// TIA Portal project "Project1" (V16)

(* hardware
DEVICE "S7-1200 station_1"  S7-1200 Station
   slot 0: "Rack_0"  S7-1200 Rack  Rack  V1.0
   slot 1: "plc_2"  CPU 1214C DC/DC/DC  6ES7 214-1AG40-0XB0  V4.4
   slot 2: "AI 4x13BIT_1"  6ES7 231-4HD32-0XB0  V2.1
   slot 3: "CB 1241 (RS485)"  CB 1241 (RS485)  6ES7 241-1CH30-1XB0  V1.0
*)

// ===== PLC "plc_2"  CPU 1214C DC/DC/DC =====

VAR_GLOBAL   // PLC tag table "Default tag table"
   "System_Byte" AT %MB1 : Byte;
   "FirstScan" AT %M1.0 : Bool;
   "DiagStatusUpdate" AT %M1.1 : Bool;
   "AlwaysTRUE" AT %M1.2 : Bool;
   "AlwaysFALSE" AT %M1.3 : Bool;
   "Clock_Byte" AT %MB0 : Byte;
   "Clock_10Hz" AT %M0.0 : Bool;
   "Clock_5Hz" AT %M0.1 : Bool;
   "Clock_2.5Hz" AT %M0.2 : Bool;
   "Clock_2Hz" AT %M0.3 : Bool;
   "Clock_1.25Hz" AT %M0.4 : Bool;
   "Clock_1Hz" AT %M0.5 : Bool;
   "Clock_0.625Hz" AT %M0.6 : Bool;
   "Clock_0.5Hz" AT %M0.7 : Bool;
   "RUNNING" AT %M8.1 : Bool;
   "ALARM" AT %M8.2 : Bool;
   "WARNING" AT %M8.3 : Bool;
   "SPEED_VFD" AT %MD10 : Real;
   "CURRENT" AT %MD14 : Real;
   "POWER" AT %MD18 : Real;
   "CARD_TEMPERATURE" AT %IW22 : Int;
   "AI1" AT %MD26 : Real;
   "AI2" AT %MD30 : Real;
   "ALARM_CODE" AT %MW2 : Int;
END_VAR

DATA_BLOCK "Data_block_1"   // DB3
{ S7_Optimized_Access := 'TRUE' }
VERSION : 0.1
   VAR RETAIN
      reference_retain : Real;
   END_VAR
   VAR
      reference_no_retain : Real;
   END_VAR
   VAR RETAIN
      reference_select : Bool;   // wybór pomiędzy zmienną zapamiętywaną po utracie zasilania a zwykłą zmienną
      start_stop_retain : Bool;
   END_VAR
   VAR
      start_stop_no_retain : Bool;
   END_VAR
   VAR RETAIN
      start_stop_select : Bool;   // wybór pomiędzy zmienną zapamiętywaną po utracie zasilania a zwykłą zmienną
   END_VAR
   VAR
      REFERENCE_TO_VFD : Real;
      START_STOP_TO_VFD : Bool;
   END_VAR
BEGIN
END_DATA_BLOCK

// folder: DANFOSS_FC_202

DATA_BLOCK "DB_1_DANFOSS_FC_202"   // DB1
{ S7_Optimized_Access := 'FALSE' }
VERSION : 0.1
   VAR
      reference : Int;
      speed_vfd : Int;
      command : Word;
      current : DInt;
      power : DInt;
      card_temperature : Int;
      AI1 : DInt;
      AI2 : DInt;
      alarm : Bool;
      warning : Bool;
      status : Array[0..15] of Bool;
      alarm_code : UInt;
      alarm_code_array_index : Int := 0;
   END_VAR
BEGIN
   // status[0] : Coil 41, TRUE - At reference, FALSE - Not at reference
   // status[1] : Coil 42, TRUE - Auto mode, FALSE - Hand mode
   // status[2] : Coil 43, TRUE - In frequency range, FALSE - Out of frequency range
   // status[3] : Coil 44, TRUE - Running, FALSE - Stopped
   // status[4] : Coil 45, Not used
   // status[5] : Coil 46, TRUE - Voltage warning, FALSE - No voltage warning
   // status[6] : Coil 47, TRUE - Current limit, FALSE - Not in current limit
   // status[7] : Coil 48, TRUE - Thermal warning, FALSE - No thermal warning
   // status[8] : Coil 33, TRUE - Control ready, FALSE - Control not ready
   // status[9] : Coil 34, TRUE - Frequency converter ready, FALSE - Frequency converter not ready
   // status[10] : Coil 35, TRUE - Safety closed, FALSE - Coasting stop
   // status[11] : Coil 36, TRUE - Alarm, FALSE - No alarm
   // status[12] : Coil 37, Not used
   // status[13] : Coil 38, Not used
   // status[14] : Coil 39, Not used
   // status[15] : Coil 40, TRUE - Warning, FALSE - No warning
END_DATA_BLOCK

// folder: System blocks/Program resources

DATA_BLOCK "IEC_Counter_0_DB"   // DB2
{ S7_Optimized_Access := 'TRUE' }
AUTHOR : Simatic
FAMILY : IEC
NAME : CNTR
VERSION : 1.0
// stored: InstanceOfName IEC_COUNTER
"IEC_COUNTER"
BEGIN
END_DATA_BLOCK

// folder: (top level)

ORGANIZATION_BLOCK "Main"   // OB1, LAD, ProgramCycle
TITLE = "Main Program Sweep (Cycle)"
{ S7_Optimized_Access := 'TRUE' }
VERSION : 0.1
   VAR_INPUT
      Initial_Call : Bool;   // Initial call of this OB
      Remanence : Bool;   // =True, if remanent data are available
   END_VAR
   VAR CONSTANT
      MODBUS_ADRESS : Int := 1;
   END_VAR
BEGIN

REGION Network 1
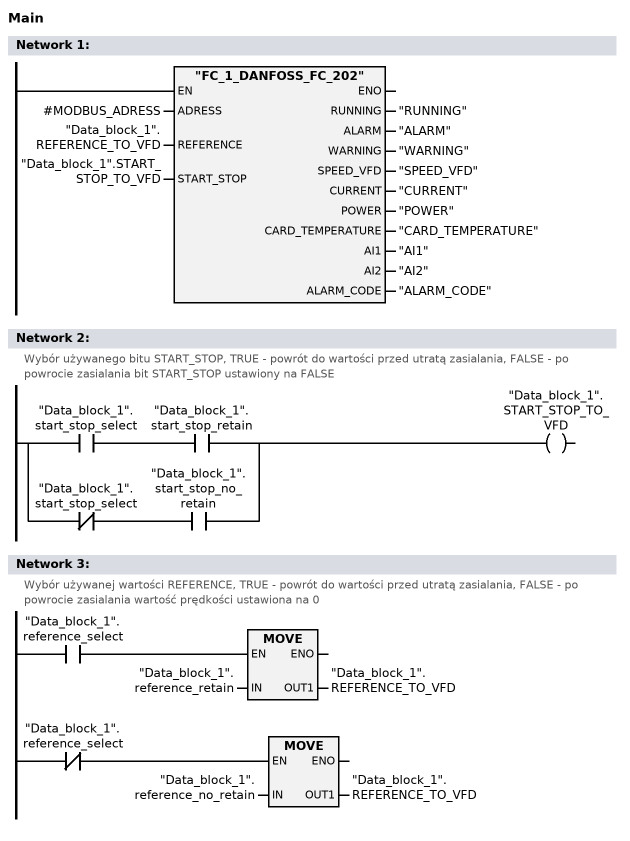
   RUNG wire#powerrail
      "FC_1_DANFOSS_FC_202"(ADRESS := #MODBUS_ADRESS, REFERENCE := "Data_block_1".REFERENCE_TO_VFD, START_STOP := "Data_block_1".START_STOP_TO_VFD, RUNNING => "RUNNING", ALARM => "ALARM", WARNING => "WARNING", SPEED_VFD => "SPEED_VFD", CURRENT => "CURRENT", POWER => "POWER", CARD_TEMPERATURE => "CARD_TEMPERATURE", AI1 => "AI1", AI2 => "AI2", ALARM_CODE => "ALARM_CODE")
   END_RUNG
   // the same network as SCL:
   "FC_1_DANFOSS_FC_202"(ADRESS := #MODBUS_ADRESS,
                         REFERENCE := "Data_block_1".REFERENCE_TO_VFD,
                         START_STOP := "Data_block_1".START_STOP_TO_VFD,
                         RUNNING => "RUNNING",
                         ALARM => "ALARM",
                         WARNING => "WARNING",
                         SPEED_VFD => "SPEED_VFD",
                         CURRENT => "CURRENT",
                         POWER => "POWER",
                         CARD_TEMPERATURE => "CARD_TEMPERATURE",
                         AI1 => "AI1",
                         AI2 => "AI2",
                         ALARM_CODE => "ALARM_CODE");
END_REGION

REGION Network 2
   // Wybór używanego bitu START_STOP, TRUE - powrót do wartości przed utratą zasialania, FALSE - po powrocie zasialania bit START_STOP ustawiony na FALSE
   RUNG wire#powerrail
      Contact( "Data_block_1".start_stop_select )
      Contact( "Data_block_1".start_stop_retain )
      wire#w1
      Coil( "Data_block_1".START_STOP_TO_VFD )
   END_RUNG
   RUNG wire#powerrail
      I_Contact( "Data_block_1".start_stop_select )
      Contact( "Data_block_1".start_stop_no_retain )
   END_RUNG wire#w1
   // the same network as SCL:
   "Data_block_1".START_STOP_TO_VFD := ("Data_block_1".start_stop_select AND "Data_block_1".start_stop_retain) OR (NOT "Data_block_1".start_stop_select AND "Data_block_1".start_stop_no_retain);
END_REGION

REGION Network 3
   // Wybór używanej wartości REFERENCE, TRUE - powrót do wartości przed utratą zasialania, FALSE - po powrocie zasialania wartość prędkości ustawiona na 0
   RUNG wire#powerrail
      Contact( "Data_block_1".reference_select )
      Move(in := "Data_block_1".reference_retain, out1 => "Data_block_1".REFERENCE_TO_VFD)
   END_RUNG
   RUNG wire#powerrail
      I_Contact( "Data_block_1".reference_select )
      Move(in := "Data_block_1".reference_no_retain, out1 => "Data_block_1".REFERENCE_TO_VFD)
   END_RUNG
   // the same network as SCL:
   IF "Data_block_1".reference_select THEN
       "Data_block_1".REFERENCE_TO_VFD := "Data_block_1".reference_retain;
   END_IF;
   IF NOT "Data_block_1".reference_select THEN
       "Data_block_1".REFERENCE_TO_VFD := "Data_block_1".reference_no_retain;
   END_IF;
END_REGION
END_ORGANIZATION_BLOCK

// folder: DANFOSS_FC_202

FUNCTION "FC_1_DANFOSS_FC_202" : Void   // FC1, LAD
{ S7_Optimized_Access := 'TRUE' }
VERSION : 0.1
   VAR_INPUT
      ADRESS : Word;   // address for the frequency converter (standard) port
      REFERENCE : Real;   // frequency 0 - 50 [Hz]
      START_STOP : Bool;   // TRUE - start, FALSE - ramp stop
   END_VAR
   VAR_OUTPUT
      RUNNING : Bool;   // TRUE - Running, FALSE - Stopped
      ALARM : Bool;   // TRUE - Alarm, FALSE - No alarm
      WARNING : Bool;   // TRUE - Warning, FALSE - No warning
      SPEED_VFD : Real;   // frequency [Hz]
      CURRENT : Real;   // current [A]
      POWER : Real;   // power [kW]
      CARD_TEMPERATURE : Int;   // control card temperarue [°C]
      AI1 : Real;   // analog input 1
      AI2 : Real;   // analog input 2
      ALARM_CODE : Int;   // the most recent logged alarm (index 0) from alarm log
   END_VAR
   VAR_TEMP
      tCommand : Word;
      tReference : Real;
      tSpeed : Real;
   END_VAR
BEGIN

REGION Network 1
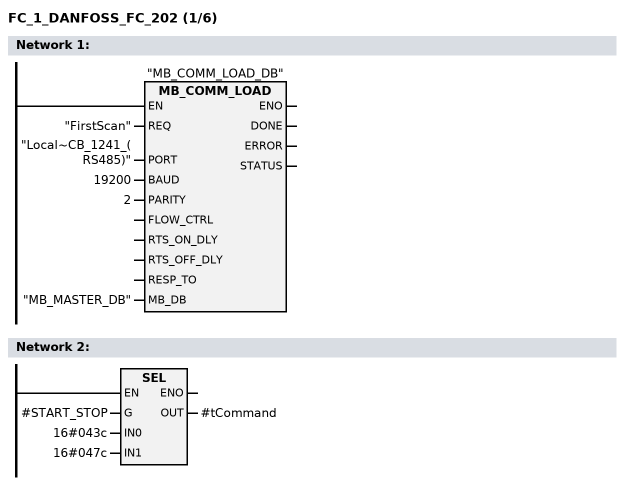
   "MB_COMM_LOAD_DB"(REQ := "FirstScan",   // MB_COMM_LOAD
                     PORT := "Local~CB_1241_(RS485)",
                     BAUD := 19200,
                     PARITY := 2,
                     MB_DB := "MB_MASTER_DB");
END_REGION

REGION Network 2
   #tCommand := SEL(G := #START_STOP, IN0 := 16#043c, IN1 := 16#047c);
END_REGION

REGION Network 3
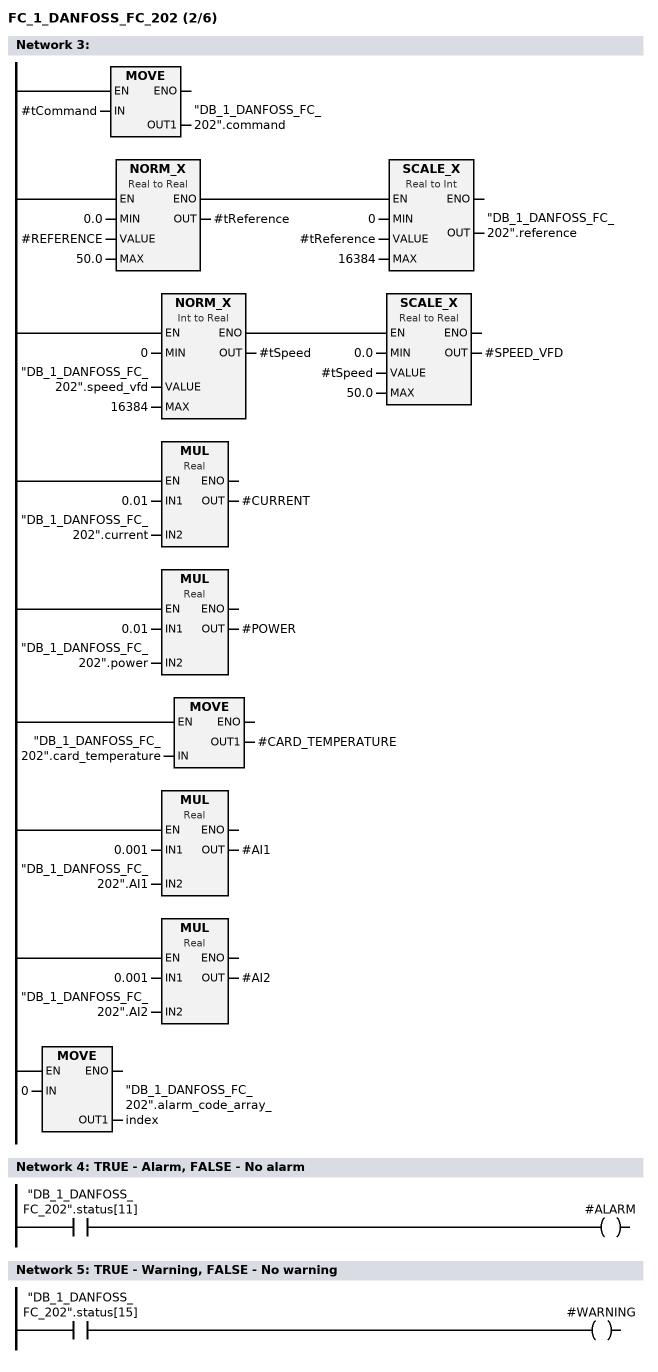
   RUNG wire#powerrail
      Move(in := #tCommand, out1 => "DB_1_DANFOSS_FC_202".command)
   END_RUNG
   RUNG wire#powerrail
      { S7_Templates := "[SrcType := Real, DestType := Real]" } Normalize(min := 0.0, value := #REFERENCE, max := 50.0, out => #tReference)
      { S7_Templates := "[SrcType := Real, DestType := Int]" } Scale(min := 0, value := #tReference, max := 16384, out => "DB_1_DANFOSS_FC_202".reference)
   END_RUNG
   RUNG wire#powerrail
      { S7_Templates := "[SrcType := Int, DestType := Real]" } Normalize(min := 0, value := "DB_1_DANFOSS_FC_202".speed_vfd, max := 16384, out => #tSpeed)
      { S7_Templates := "[SrcType := Real, DestType := Real]" } Scale(min := 0.0, value := #tSpeed, max := 50.0, out => #SPEED_VFD)
   END_RUNG
   RUNG wire#powerrail
      { S7_Templates := "SrcType := Real" } Mul(in1 := 0.01, in2 := "DB_1_DANFOSS_FC_202".current, out => #CURRENT)
   END_RUNG
   RUNG wire#powerrail
      { S7_Templates := "SrcType := Real" } Mul(in1 := 0.01, in2 := "DB_1_DANFOSS_FC_202".power, out => #POWER)
   END_RUNG
   RUNG wire#powerrail
      Move(in := "DB_1_DANFOSS_FC_202".card_temperature, out1 => #CARD_TEMPERATURE)
   END_RUNG
   RUNG wire#powerrail
      { S7_Templates := "SrcType := Real" } Mul(in1 := 0.001, in2 := "DB_1_DANFOSS_FC_202".AI1, out => #AI1)
   END_RUNG
   RUNG wire#powerrail
      { S7_Templates := "SrcType := Real" } Mul(in1 := 0.001, in2 := "DB_1_DANFOSS_FC_202".AI2, out => #AI2)
   END_RUNG
   RUNG wire#powerrail
      Move(in := 0, out1 => "DB_1_DANFOSS_FC_202".alarm_code_array_index)
   END_RUNG
   // the same network as SCL:
   "DB_1_DANFOSS_FC_202".command := #tCommand;
   #tReference := NORM_X(MIN := 0.0, VALUE := #REFERENCE, MAX := 50.0);
   "DB_1_DANFOSS_FC_202".reference := SCALE_X(MIN := 0, VALUE := #tReference, MAX := 16384);
   #tSpeed := NORM_X(MIN := 0, VALUE := "DB_1_DANFOSS_FC_202".speed_vfd, MAX := 16384);
   #SPEED_VFD := SCALE_X(MIN := 0.0, VALUE := #tSpeed, MAX := 50.0);
   #CURRENT := 0.01 * "DB_1_DANFOSS_FC_202".current;
   #POWER := 0.01 * "DB_1_DANFOSS_FC_202".power;
   #CARD_TEMPERATURE := "DB_1_DANFOSS_FC_202".card_temperature;
   #AI1 := 0.001 * "DB_1_DANFOSS_FC_202".AI1;
   #AI2 := 0.001 * "DB_1_DANFOSS_FC_202".AI2;
   "DB_1_DANFOSS_FC_202".alarm_code_array_index := 0;
END_REGION

REGION Network 4: TRUE - Alarm, FALSE - No alarm
   RUNG wire#powerrail
      Contact( "DB_1_DANFOSS_FC_202".status[11] )
      Coil( #ALARM )
   END_RUNG
   // the same network as SCL:
   #ALARM := "DB_1_DANFOSS_FC_202".status[11];
END_REGION

REGION Network 5: TRUE - Warning, FALSE - No warning
   RUNG wire#powerrail
      Contact( "DB_1_DANFOSS_FC_202".status[15] )
      Coil( #WARNING )
   END_RUNG
   // the same network as SCL:
   #WARNING := "DB_1_DANFOSS_FC_202".status[15];
END_REGION

REGION Network 6
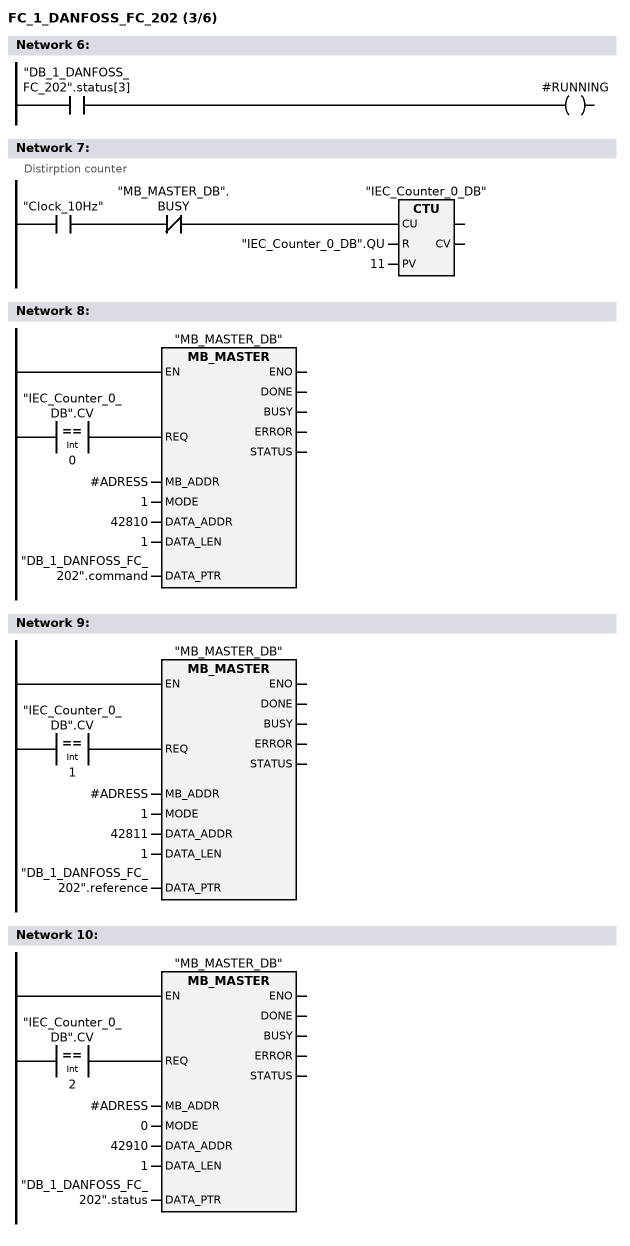
   RUNG wire#powerrail
      Contact( "DB_1_DANFOSS_FC_202".status[3] )
      Coil( #RUNNING )
   END_RUNG
   // the same network as SCL:
   #RUNNING := "DB_1_DANFOSS_FC_202".status[3];
END_REGION

REGION Network 7
   // Distirption counter
   "IEC_Counter_0_DB".CTU(CU := "Clock_10Hz" AND NOT "MB_MASTER_DB".BUSY, R := "IEC_Counter_0_DB".QU, PV := 11);
END_REGION

REGION Network 8
   "MB_MASTER_DB"(REQ := "IEC_Counter_0_DB".CV = 0,   // MB_MASTER
                  MB_ADDR := #ADRESS,
                  MODE := 1,
                  DATA_ADDR := 42810,
                  DATA_LEN := 1,
                  DATA_PTR := "DB_1_DANFOSS_FC_202".command);
END_REGION

REGION Network 9
   "MB_MASTER_DB"(REQ := "IEC_Counter_0_DB".CV = 1,   // MB_MASTER
                  MB_ADDR := #ADRESS,
                  MODE := 1,
                  DATA_ADDR := 42811,
                  DATA_LEN := 1,
                  DATA_PTR := "DB_1_DANFOSS_FC_202".reference);
END_REGION

REGION Network 10
   "MB_MASTER_DB"(REQ := "IEC_Counter_0_DB".CV = 2,   // MB_MASTER
                  MB_ADDR := #ADRESS,
                  MODE := 0,
                  DATA_ADDR := 42910,
                  DATA_LEN := 1,
                  DATA_PTR := "DB_1_DANFOSS_FC_202".status);
END_REGION

REGION Network 11
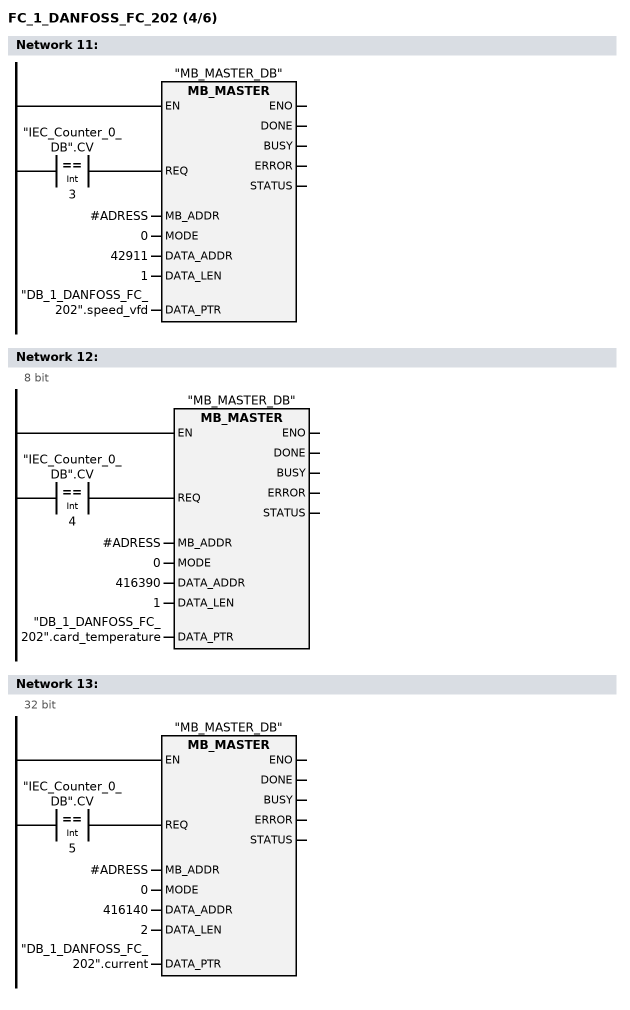
   "MB_MASTER_DB"(REQ := "IEC_Counter_0_DB".CV = 3,   // MB_MASTER
                  MB_ADDR := #ADRESS,
                  MODE := 0,
                  DATA_ADDR := 42911,
                  DATA_LEN := 1,
                  DATA_PTR := "DB_1_DANFOSS_FC_202".speed_vfd);
END_REGION

REGION Network 12
   // 8 bit
   "MB_MASTER_DB"(REQ := "IEC_Counter_0_DB".CV = 4,   // MB_MASTER
                  MB_ADDR := #ADRESS,
                  MODE := 0,
                  DATA_ADDR := 416390,
                  DATA_LEN := 1,
                  DATA_PTR := "DB_1_DANFOSS_FC_202".card_temperature);
END_REGION

REGION Network 13
   // 32 bit
   "MB_MASTER_DB"(REQ := "IEC_Counter_0_DB".CV = 5,   // MB_MASTER
                  MB_ADDR := #ADRESS,
                  MODE := 0,
                  DATA_ADDR := 416140,
                  DATA_LEN := 2,
                  DATA_PTR := "DB_1_DANFOSS_FC_202".current);
END_REGION

REGION Network 14
   // 32 bit
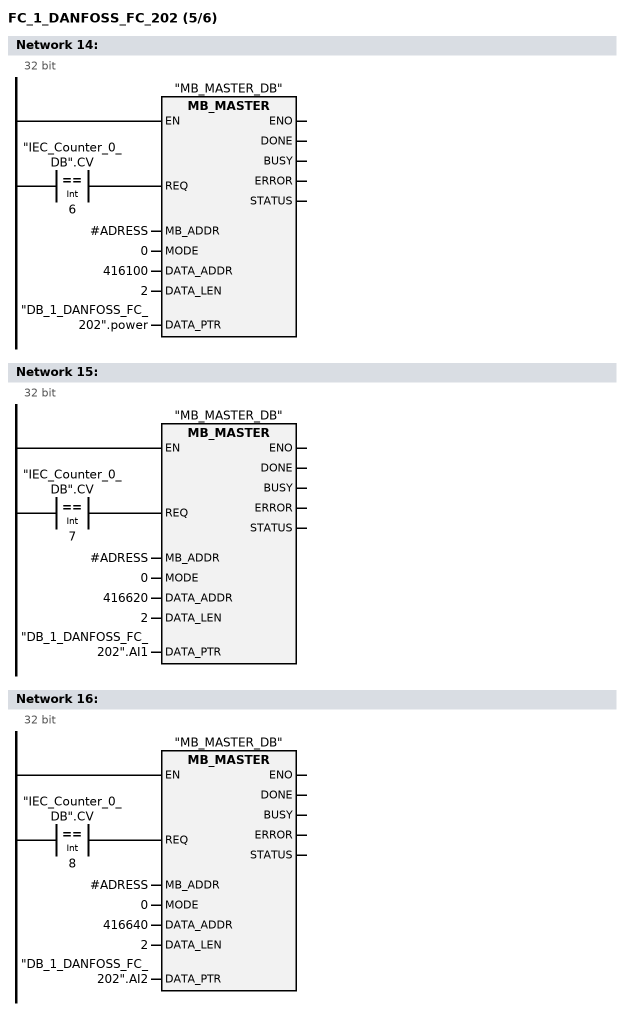
   "MB_MASTER_DB"(REQ := "IEC_Counter_0_DB".CV = 6,   // MB_MASTER
                  MB_ADDR := #ADRESS,
                  MODE := 0,
                  DATA_ADDR := 416100,
                  DATA_LEN := 2,
                  DATA_PTR := "DB_1_DANFOSS_FC_202".power);
END_REGION

REGION Network 15
   // 32 bit
   "MB_MASTER_DB"(REQ := "IEC_Counter_0_DB".CV = 7,   // MB_MASTER
                  MB_ADDR := #ADRESS,
                  MODE := 0,
                  DATA_ADDR := 416620,
                  DATA_LEN := 2,
                  DATA_PTR := "DB_1_DANFOSS_FC_202".AI1);
END_REGION

REGION Network 16
   // 32 bit
   "MB_MASTER_DB"(REQ := "IEC_Counter_0_DB".CV = 8,   // MB_MASTER
                  MB_ADDR := #ADRESS,
                  MODE := 0,
                  DATA_ADDR := 416640,
                  DATA_LEN := 2,
                  DATA_PTR := "DB_1_DANFOSS_FC_202".AI2);
END_REGION

REGION Network 17
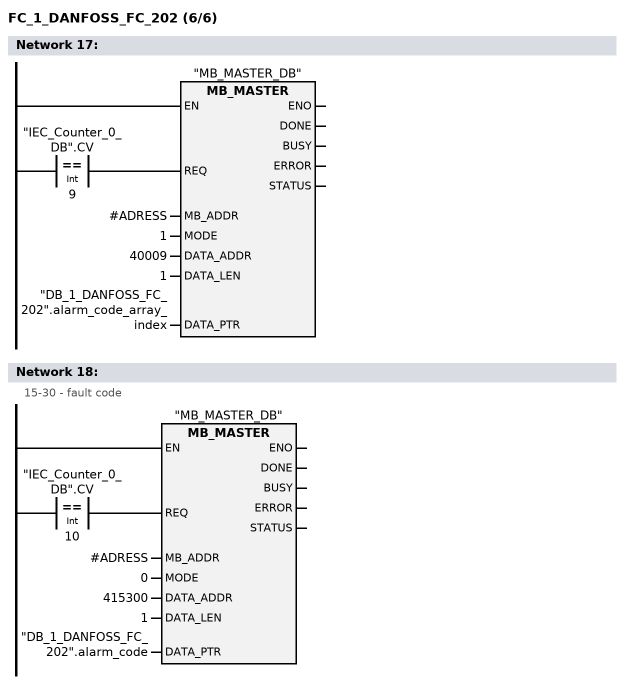
   "MB_MASTER_DB"(REQ := "IEC_Counter_0_DB".CV = 9,   // MB_MASTER
                  MB_ADDR := #ADRESS,
                  MODE := 1,
                  DATA_ADDR := 40009,
                  DATA_LEN := 1,
                  DATA_PTR := "DB_1_DANFOSS_FC_202".alarm_code_array_index);
END_REGION

REGION Network 18
   // 15-30 - fault code
   "MB_MASTER_DB"(REQ := "IEC_Counter_0_DB".CV = 10,   // MB_MASTER
                  MB_ADDR := #ADRESS,
                  MODE := 0,
                  DATA_ADDR := 415300,
                  DATA_LEN := 1,
                  DATA_PTR := "DB_1_DANFOSS_FC_202".alarm_code);
END_REGION
END_FUNCTION